INTERFACE I_StringBuilder

METHOD M_Append : I_StringBuilder
VAR_INPUT
	Value	: STRING(255);
END_VAR
END_METHOD

METHOD PUBLIC M_AppendBOOL  : I_StringBuilder
VAR_INPUT
	Value:			BOOL;
END_VAR
END_METHOD

METHOD PUBLIC M_AppendINT : I_StringBuilder
VAR_INPUT
	Value	: LINT;
END_VAR
END_METHOD

METHOD PUBLIC M_AppendREAL : I_StringBuilder
VAR_INPUT
	Value:		LREAL;
	Decimals:	SINT;
END_VAR
END_METHOD

METHOD PUBLIC M_Contains : BOOL
VAR_INPUT
	Value	: STRING(255);
END_VAR
END_METHOD

METHOD M_Find : UDINT
VAR_INPUT
	Value	: STRING(255);
END_VAR
END_METHOD

METHOD M_Insert : I_StringBuilder
VAR_INPUT
	Position:	UDINT;
	Value:		STRING(255);
END_VAR
END_METHOD

METHOD M_Remove : I_StringBuilder
VAR_INPUT
	Position:	UDINT;
	Length:		UDINT;
END_VAR
END_METHOD

METHOD M_Replace : I_StringBuilder
VAR_INPUT
	Target:		STRING(255);
	Value:		STRING(255);
END_VAR
END_METHOD

METHOD M_Reset : I_StringBuilder
END_METHOD

METHOD M_ToAny : BOOL
VAR_INPUT
	Value:			ANY_STRING;
END_VAR
END_METHOD

METHOD PUBLIC M_ToString : String(255)
VAR_INPUT
END_VAR
END_METHOD

PROPERTY PUBLIC P_Length : Udint
GET
END_GET
END_PROPERTY

END_INTERFACE

(* stored: Version 1.1.0.1
   Itf I_StringBuilder: Id {df3d4a37-6b19-0224-3a23-50c560e48de6}
   Method M_Append: Id {ba3dc35a-00e3-0c07-0dfd-8c13ef431e5e}
   Method M_AppendBOOL: Id {7603f41d-77e0-0877-3137-edeb0957466d}
   Method M_AppendINT: Id {14f51f13-e329-0cde-0c9e-a7dc465a3499}
   Method M_AppendREAL: Id {f057156e-5dae-0fd8-10fe-cc573cd3ed43}
   Method M_Contains: Id {74317bae-5e12-0a37-3a16-0b339f34807e}
   Method M_Find: Id {1f3e8d49-9a77-09ce-067b-462519976714}
   Method M_Insert: Id {a5a38218-1f4c-01ff-2b1b-ab5893013608}
   Method M_Remove: Id {76d21321-4b15-00ee-14ed-3c5f85060525}
   Method M_Replace: Id {b6703233-b9c6-04c9-1787-fcb0a8311196}
   Method M_Reset: Id {c51c1de9-e242-0e2e-15b4-007d70478885}
   Method M_ToAny: Id {940c2d63-a99a-009b-232c-ea17ccc23948}
   Method M_ToString: Id {3d41c117-e4c2-0981-0e95-35260077a987}
   Property P_Length: Id {917505ca-54ce-03d7-1d45-2467135a7e41}
   Get Get: Id {9df562a0-8d74-0cfe-38db-8a1fcfe61f0c} *)
